Yaskawa INFORM job: R1_W17,20,22(0,0)OK-KMNEW.JBI

/JOB
//NAME R1_W17,20,22(0,0)OK-KMNEW
///FOLDERNAME KRIS-SCIANA
//POS
///NPOS 166,166,0,10,0,0
///TOOL 0
///POSTYPE PULSE
///PULSE
C00000=-143433,-90175,-75020,-14586,83972,33032
C00001=-153732,-78635,-58192,-14050,77869,30109
C00002=-157098,-74863,-52692,-13875,75874,29154
C00003=-157098,-74243,-51213,-13910,75301,29220
C00004=-157098,-74333,-51423,-13906,75382,29211
C00005=-158949,-72964,-50795,-13730,75376,28555
C00006=-157200,-74632,-52271,-13875,75723,29138
C00007=-211231,-129831,-71825,-7304,52478,11413
C00008=-211231,-128371,-70027,-7339,52125,11439
C00009=-211231,-126878,-68176,-7377,51757,11467
C00010=-211231,-127047,-68387,-7373,51799,11463
C00011=-212771,-124423,-67855,-6939,52685,10797
C00012=-211231,-128089,-69679,-7347,52057,11444
C00013=-232444,-132787,-72439,-2403,50152,3160
C00014=-232444,-131349,-70721,-2414,49837,3167
C00015=-232444,-129731,-68771,-2422,49470,3172
C00016=-232444,-129852,-68917,-2422,49498,3172
C00017=-232842,-127642,-68505,-2293,50368,2994
C00018=-232444,-131710,-71149,-2407,49917,3162
C00019=-145968,-32886,-32033,-14386,86409,31863
C00020=-145968,-32298,-29296,-14401,85068,32019
C00021=-145968,-31942,-27784,-14425,84347,32104
C00022=-145968,-31980,-27951,-14410,84425,32095
C00023=-147178,-31176,-27384,-14348,84275,31690
C00024=-145968,-32285,-29241,-14400,85043,32023
C00025=-139425,14039,5691,-14754,88455,33906
C00026=-139519,13379,6497,-14751,87629,33972
C00027=-139519,13616,7680,-14752,87041,34041
C00028=-139519,13563,7430,-14752,87165,34026
C00029=-140335,14099,7919,-14713,86994,33760
C00030=-140218,14798,7500,-14716,87614,33729
C00031=-139869,18363,10790,-14729,87489,33867
C00032=-140218,14798,7500,-14716,87614,33729
C00033=-140402,1849,-19527,-14902,97240,32509
C00034=-140435,1808,-19560,-14885,97235,32499
C00035=-142735,10961,1802,-14568,88645,32727
C00036=-142735,11930,7018,-14580,86016,33037
C00037=-142735,12205,8255,-14585,85414,33107
C00038=-142735,12159,8055,-14585,85510,33096
C00039=-143548,12776,8612,-14541,85338,32830
C00040=-143548,12478,7250,-14533,86001,32752
C00041=-142989,17280,11639,-14579,85875,32965
C00042=-143548,12478,7250,-14533,86001,32752
C00043=-153871,-49826,-39465,-13916,81020,29711
C00044=-153871,-49427,-38150,-13936,80432,29777
C00045=-153871,-48844,-36293,-13969,79619,29871
C00046=-153871,-48918,-36516,-13965,79718,29861
C00047=-155772,-47404,-35637,-13806,79621,29203
C00048=-153871,-49375,-37964,-13941,80356,29788
C00049=-176442,-83720,-50224,-26100,86167,24219
C00050=-176268,-83127,-48832,-26086,85723,24382
C00051=-176268,-82702,-48032,-26088,85476,24434
C00052=-176268,-82805,-48225,-26088,85536,24421
C00053=-177470,-81547,-47714,-26247,85464,23996
C00054=-176268,-83563,-49657,-26078,85980,24323
C00055=-152058,-57095,-47355,-15849,91689,31553
C00056=-147010,-10638,-8183,-21391,105329,31267
C00057=-140743,-13850,-3598,-31425,97214,46819
C00058=-163982,-90504,-45918,-34963,77070,43608
C00059=-165644,-92905,-46739,-35256,75820,43353
C00060=-158551,-98871,-68851,-16167,82483,30472
C00061=-139863,-9121,-22514,-12675,86754,36604
C00062=-142907,-1645,-8358,-12312,81526,36078
C00063=-137448,8074,8661,-24597,77704,52502
C00064=-134515,54764,60771,-29890,95701,49675
C00065=-140743,-13850,-3598,-31425,97214,46819
C00066=-146433,-61661,-62839,-14679,91621,33634
C00067=-152691,-57358,-64796,-14380,93822,31204
C00068=-159687,-62193,-51187,-13527,81199,28324
C00069=-149187,-17486,-8424,-28072,102983,37207
C00070=-171257,-77817,-43106,-31829,86773,32910
C00071=-172558,-79550,-43833,-32051,85919,32654
C00072=-179422,-87952,-47149,-33191,81425,31301
C00073=-188034,-95777,-49870,-34529,76186,29541
C00074=-201576,-85135,-50180,-27119,84644,21010
C00075=-189185,-159173,-100064,-12251,58132,22119
C00076=-139628,-22178,-29745,-13339,88451,36438
C00077=-142464,16713,5801,-14603,90978,35100
C00078=-140096,48315,46031,-21206,94479,42259
C00079=-138998,70596,76957,-24600,99628,41883
C00080=-149221,-17459,-8404,-28081,102973,37195
C00081=-142912,-78923,-74681,-14594,91271,34909
C00082=96,-41537,-55485,-8102,54341,61135
C00083=96,-41537,-55485,-8102,54341,61135
C00084=-47991,-26757,-28892,6367,80786,-11975
C00085=-57126,-9114,2182,8032,71615,-15703
C00086=-56289,-5858,6360,8073,70774,-15813
C00087=-54160,-1963,12621,8049,68923,-15724
C00088=-54160,-1355,14168,8081,68290,-15768
C00089=-54160,-1431,13975,8077,68369,-15762
C00090=-53417,516,15594,7965,68299,-15502
C00091=-53699,-1671,12330,7961,69203,-15542
C00092=-56482,3777,16911,8368,69462,-16522
C00093=-53699,-1671,12330,7961,69203,-15542
C00094=-16096,-40309,-15630,1558,64307,-2146
C00095=-15667,-39835,-14323,1484,63739,-1996
C00096=-15667,-38980,-12408,1491,63001,-2002
C00097=-15667,-39089,-12651,1491,63095,-2002
C00098=-15228,-35710,-10538,1402,63524,-1836
C00099=-15475,-38012,-12587,1447,63607,-1924
C00100=26525,-36306,-13799,-6251,66511,13302
C00101=27157,-34792,-10896,-6403,65558,13584
C00102=27157,-34039,-9183,-6437,64895,13622
C00103=27157,-34142,-9408,-6432,64981,13617
C00104=26710,-32142,-8110,-6346,65173,13444
C00105=27121,-34968,-11568,-6383,65877,13555
C00106=38673,-31750,-14829,-8018,70533,17427
C00107=38106,-27047,-6323,-8075,67686,17416
C00108=38106,-26024,-3889,-8132,66720,17484
C00109=38106,-26093,-4052,-8129,66783,17480
C00110=37587,-24395,-2874,-8044,66879,17284
C00111=38095,-27443,-7349,-8055,68105,17383
C00112=33691,-40237,-37529,-4343,78333,9389
C00113=4088,-38479,-36421,-4266,78531,9229
C00114=6240,-59965,-30493,-1746,62990,4256
C00115=6240,-59198,-28889,-1752,62394,4263
C00116=6240,-59277,-29056,-1752,62455,4263
C00117=6137,-57545,-28162,-1726,62793,4220
C00118=6137,-58794,-30830,-1711,63793,4205
C00119=1139,-59118,-30998,-730,63654,2372
C00120=6137,-58794,-30830,-1711,63793,4205
C00121=47807,-38519,-19261,-8869,69876,19011
C00122=47539,-37304,-17377,-8859,69317,18957
C00123=47539,-36567,-15561,-8901,68588,19011
C00124=47539,-36658,-15781,-8894,68676,19004
C00125=47029,-35461,-15018,-8811,68766,18813
C00126=47893,-38902,-19858,-8871,70056,19027
C00127=73069,7126,14309,-11765,75874,27473
C00128=72335,9424,18352,-11759,74488,27349
C00129=72335,9956,19820,-11792,73873,27410
C00130=72335,9884,19621,-11787,73955,27403
C00131=71491,11415,20993,-11706,73779,27121
C00132=71657,3792,9684,-11575,76785,26891
C00133=61085,-36100,-21666,6391,58079,18912
C00134=49069,-45805,-25229,-7304,68786,15386
C00135=19871,-63611,-22023,35378,44606,-3365
C00136=17766,-52406,-14755,34280,50845,-2144
C00137=56335,-20769,8067,22753,38631,7110
C00138=59032,-16534,11142,20917,38204,8486
C00139=60031,-14754,12465,20223,38057,9000
C00140=61085,-36100,-21666,6391,58079,18912
C00141=29040,-81101,-50034,-3867,64562,8354
C00142=7217,-74366,-42042,361,62632,377
C00143=-16654,-66617,-25209,25593,50854,-13543
C00144=-27368,-47601,-12216,38001,70169,-15327
C00145=17766,-52406,-14755,34280,50845,-2144
C00146=46390,-61269,-41061,-6756,70352,14356
C00147=42236,-65961,-43421,-6101,69070,12939
C00148=21298,-49858,-1802,32067,40583,-8230
C00149=20826,-44930,4480,33075,39613,-8917
C00150=60671,-13467,25003,8839,33164,11366
C00151=62121,-10887,26961,7730,33147,12189
C00152=66302,-2318,33759,4536,33070,14551
C00153=69057,3829,38920,2429,32943,16104
C00154=60086,17396,47844,26002,45227,9224
C00155=60912,19537,49876,25778,44850,9513
C00156=60912,14444,39766,24345,48130,10454
C00157=78652,23072,35845,-11228,70256,25748
C00158=41637,-60211,-42225,-5828,71489,12454
C00159=-9438,-58348,-23745,3601,60262,-5968
C00160=-15357,-59811,-7616,12634,36711,-18275
C00161=-36406,-36757,8811,38530,63422,-26409
C00162=20826,-44930,4480,33075,39613,-8917
C00163=27379,-50240,-5351,20739,41756,-1745
C00164=50643,-51074,-27069,-7729,67873,16514
C00165=-88506,-94181,-91931,-709,81235,59832
BC00000=335653,8129,711615
BC00001=335653,8129,711615
BC00002=335653,8129,711615
BC00003=335653,8129,711615
BC00004=335653,8129,711615
BC00005=335653,8129,711615
BC00006=335653,8129,711615
BC00007=335653,8130,711613
BC00008=335653,8130,711613
BC00009=335653,8130,711613
BC00010=335653,8130,711613
BC00011=335653,8130,711613
BC00012=335653,8130,711613
BC00013=335653,1154,711613
BC00014=335653,1155,711613
BC00015=335653,1155,711613
BC00016=335653,1155,711613
BC00017=335653,1155,711613
BC00018=335653,1155,711613
BC00019=335653,1154,711612
BC00020=335653,1154,711612
BC00021=335653,1154,711612
BC00022=335653,1154,711612
BC00023=335653,1154,711612
BC00024=335653,1154,711612
BC00025=335653,1152,711610
BC00026=335653,1152,711610
BC00027=335653,1152,711610
BC00028=335653,1152,711610
BC00029=335653,1152,711610
BC00030=335653,1152,711610
BC00031=335653,1152,711610
BC00032=335653,1152,711610
BC00033=335653,1152,711610
BC00034=160380,1151,711608
BC00035=160380,1151,715049
BC00036=160380,1151,715049
BC00037=160380,1151,715049
BC00038=160380,1151,715049
BC00039=160380,1151,715049
BC00040=160380,1151,715049
BC00041=160380,1152,715048
BC00042=160380,1151,715049
BC00043=160380,1151,715049
BC00044=160380,1151,715049
BC00045=160380,1151,715049
BC00046=160380,1151,715049
BC00047=160380,1151,715049
BC00048=160380,1151,715049
BC00049=160380,1151,715049
BC00050=160380,1151,715049
BC00051=160380,1151,715049
BC00052=160380,1151,715049
BC00053=160380,1151,715049
BC00054=160380,1151,715049
BC00055=160380,1151,715049
BC00056=160380,1151,715049
BC00057=160380,1151,715049
BC00058=160380,1151,715049
BC00059=160380,1151,715049
BC00060=160381,1151,715048
BC00061=160381,1151,715048
BC00062=160381,1151,715048
BC00063=160382,1151,715048
BC00064=160382,1151,715048
BC00065=160380,1151,715049
BC00066=160381,1151,715048
BC00067=347379,1151,715048
BC00068=347379,1151,715048
BC00069=347378,1151,715047
BC00070=347378,1151,715047
BC00071=347378,1151,715047
BC00072=347378,1151,715046
BC00073=347378,1151,715046
BC00074=347378,1151,715046
BC00075=347379,1151,715048
BC00076=347379,1151,715048
BC00077=347379,1151,715048
BC00078=347378,1151,715047
BC00079=347378,1151,715047
BC00080=347378,1151,715047
BC00081=347379,1151,715048
BC00082=71294,1151,1035267
BC00083=71294,1151,1035267
BC00084=14908,77377,861464
BC00085=14908,77377,833834
BC00086=14908,77377,833863
BC00087=14909,77377,833909
BC00088=14909,77377,833909
BC00089=14909,77377,833909
BC00090=14909,77377,833909
BC00091=14909,77377,833909
BC00092=14909,77377,833909
BC00093=14909,77377,833909
BC00094=14909,77377,833909
BC00095=14909,77377,833909
BC00096=14909,77376,833908
BC00097=14909,77376,833908
BC00098=14909,77376,833908
BC00099=14909,77376,833908
BC00100=14909,77376,833908
BC00101=14909,77376,833908
BC00102=14909,77376,833908
BC00103=14909,77376,833908
BC00104=14909,77376,833908
BC00105=14909,77376,833908
BC00106=14909,77376,833908
BC00107=14909,77376,833908
BC00108=14909,77376,833907
BC00109=14909,77376,833907
BC00110=14909,77376,833907
BC00111=14909,77376,833907
BC00112=14908,77377,833834
BC00113=166638,196652,833834
BC00114=218128,196652,810863
BC00115=218128,196652,810863
BC00116=218128,196652,810863
BC00117=218128,196652,810863
BC00118=218128,196652,810863
BC00119=218128,196652,810863
BC00120=218128,196652,810863
BC00121=218128,196652,810863
BC00122=218128,196652,810863
BC00123=218128,196652,810863
BC00124=218128,196652,810863
BC00125=218128,196652,810863
BC00126=218128,196652,810863
BC00127=218127,196651,810862
BC00128=218127,196651,810862
BC00129=218127,196651,810862
BC00130=218127,196651,810862
BC00131=218127,196651,810862
BC00132=218127,196651,810862
BC00133=218128,196652,810863
BC00134=218128,196652,810863
BC00135=218128,196652,810863
BC00136=218128,196652,810863
BC00137=218128,196652,810863
BC00138=218128,196652,810863
BC00139=218128,196652,810863
BC00140=218128,196652,810863
BC00141=218128,196652,810863
BC00142=218128,196652,810863
BC00143=218128,196652,810863
BC00144=218128,196652,810863
BC00145=218128,196652,810863
BC00146=218128,196652,810863
BC00147=35771,188457,887876
BC00148=35771,188457,887876
BC00149=35771,188457,887876
BC00150=35771,188457,887876
BC00151=35771,188457,887876
BC00152=35771,188457,887876
BC00153=35771,188457,887876
BC00154=35771,188457,887876
BC00155=35771,188457,887876
BC00156=35771,188457,887876
BC00157=35772,185483,887872
BC00158=35772,185483,887872
BC00159=35772,185483,887872
BC00160=35771,188457,887876
BC00161=35771,188457,887876
BC00162=35771,188457,887876
BC00163=36231,187575,887592
BC00164=38104,183984,886436
BC00165=294911,15771,909309
///POSTYPE BASE
///RECTAN
///RCONF 0,0,0,0,1,0,0,0,0,0,0,0,0,0,0,0,0,0,0,0,0,0,0,0
P00006=2.006,1.622,-0.565,0.0000,0.0000,0.0000
P00021=0.073,2.058,-0.109,0.0000,0.0000,0.0000
P00022=2.006,1.622,-0.565,0.0000,0.0000,0.0000
///RCONF 0,0,0,0,0,0,0,0,0,0,0,0,0,0,0,0,0,0,0,0,0,0,0,0
P00023=-2.957,-4.083,2.762,0.0000,0.0000,0.0000
P00024=-1.466,-0.226,-0.419,0.0000,0.0000,0.0000
P00025=3.643,0.007,-2.585,0.0000,0.0000,0.0000
P00026=2.644,0.055,-2.583,0.0000,0.0000,0.0000
P00027=2.278,0.099,-4.210,0.0000,0.0000,0.0000
P00028=-1.778,-0.182,-2.050,0.0000,0.0000,0.0000
P00029=1.749,4.006,-0.261,0.0000,0.0000,0.0000
//INST
///DATE 2025/04/16 06:31
///ATTR SC,RW
///GROUP1 RB1,BS1
///LVARS 0,1,0,0,0,2,2,0
NOP
MOVJ C00000 BC00000 VJ=50.00
SFTOF
MOVL C00001 BC00001 V=333.3
MOVL C00002 BC00002 V=166.7
REFP 3 C00003 BC00003
CALL JOB:SEARCH-R1
SET P021 P006
SFTON P021
MOVL C00004 BC00004 V=60.0
REFP 3 C00005 BC00005
CALL JOB:SEARCH-R1
SET P021 P006
SFTON P021
MOVL C00006 BC00006 V=166.7
MOVL C00007 BC00007 V=500.0
MOVL C00008 BC00008 V=166.7
REFP 3 C00009 BC00009
CALL JOB:SEARCH-R1
SET P022 P006
SFTON P022
MOVL C00010 BC00010 V=60.0
REFP 3 C00011 BC00011
CALL JOB:SEARCH-R1
SET P022 P006
SFTON P022
MOVL C00012 BC00012 V=166.7
MOVL C00013 BC00013 V=500.0
MOVL C00014 BC00014 V=166.7
REFP 3 C00015 BC00015
CALL JOB:SEARCH-R1
SET P023 P006
SFTON P023
MOVL C00016 BC00016 V=60.0
REFP 3 C00017 BC00017
CALL JOB:SEARCH-R1
SET P023 P006
SFTON P023
MOVL C00018 BC00018 V=166.7
MOVL C00019 BC00019 V=500.0
MOVL C00020 BC00020 V=166.7
REFP 3 C00021 BC00021
CALL JOB:SEARCH-R1
SET P024 P006
SFTON P024
MOVL C00022 BC00022 V=60.0
REFP 3 C00023 BC00023
CALL JOB:SEARCH-R1
SET P024 P006
SFTON P024
MOVL C00024 BC00024 V=166.7
MOVL C00025 BC00025 V=500.0
MOVL C00026 BC00026 V=166.7
REFP 3 C00027 BC00027
CALL JOB:SEARCH-R1
SET P025 P006
SFTON P025
MOVL C00028 BC00028 V=60.0
REFP 3 C00029 BC00029
CALL JOB:SEARCH-R1
SET P025 P006
SFTON P025
MOVL C00030 BC00030 V=166.7
REFP 3 C00031 BC00031
CALL JOB:SEARCH-R1
SET P025 P006
SFTON P025
MOVL C00032 BC00032 V=166.7
SFTOF
MOVL C00033 BC00033 V=500.0
MOVL C00034 BC00034 V=500.0
MOVL C00035 BC00035 V=500.0
MOVL C00036 BC00036 V=166.7
REFP 3 C00037 BC00037
CALL JOB:SEARCH-R1
SET P026 P006
SFTON P026
MOVL C00038 BC00038 V=60.0
REFP 3 C00039 BC00039
CALL JOB:SEARCH-R1
SET P026 P006
SFTON P026
MOVL C00040 BC00040 V=166.7
REFP 3 C00041 BC00041
CALL JOB:SEARCH-R1
SET P026 P006
SFTON P026
MOVL C00042 BC00042 V=166.7
MOVL C00043 BC00043 V=500.0
MOVL C00044 BC00044 V=166.7
REFP 3 C00045 BC00045
CALL JOB:SEARCH-R1
SET P027 P006
SFTON P027
MOVL C00046 BC00046 V=60.0
REFP 3 C00047 BC00047
CALL JOB:SEARCH-R1
SET P027 P006
SFTON P027
MOVL C00048 BC00048 V=166.7
MOVL C00049 BC00049 V=500.0
MOVL C00050 BC00050 V=166.7
REFP 3 C00051 BC00051
CALL JOB:SEARCH-R1
SET P028 P006
SFTON P028
MOVL C00052 BC00052 V=60.0
REFP 3 C00053 BC00053
CALL JOB:SEARCH-R1
SET P028 P006
SFTON P028
MOVL C00054 BC00054 V=166.7
SFTOF
MOVL C00055 BC00055 V=166.7
CALL JOB:COFNIJ_DRUT
MACRO1 MJ#(0) ARGF9
MOVL C00056 BC00056 V=500.0
SFTON P027
MOVL C00057 BC00057 V=166.7 PL=0
ARCON
SFTON P028
MOVL C00058 BC00058 V=12.5
MOVL C00059 BC00059 V=12.5
ARCOF
SFTOF
MOVJ C00060 BC00060 VJ=25.00
MOVJ C00061 BC00061 VJ=25.00
MOVJ C00062 BC00062 VJ=25.00
SFTON P026
MOVL C00063 BC00063 V=166.7 PL=0
ARCON
MOVL C00064 BC00064 V=12.5
SFTON P027
MOVL C00065 BC00065 V=12.5
ARCOF
SFTOF
MOVJ C00066 BC00066 VJ=25.00
MOVJ C00067 BC00067 VJ=25.00
MOVJ C00068 BC00068 VJ=25.00
SFTON P021
MOVL C00069 BC00069 V=166.7 PL=0
ARCON
SFTON P022
MOVL C00070 BC00070 V=12.5
MOVL C00071 BC00071 V=12.5
ARCOF
SFTON P023
MOVL C00072 BC00072 V=41.7 PL=0
ARCON
MOVL C00073 BC00073 V=12.5
MOVL C00074 BC00074 V=12.5
ARCOF
SFTOF
MOVJ C00075 BC00075 VJ=25.00
MOVJ C00076 BC00076 VJ=25.00
MOVJ C00077 BC00077 VJ=25.00
SFTON P024
MOVL C00078 BC00078 V=166.7 PL=0
ARCON
MOVL C00079 BC00079 V=12.5
SFTON P021
MOVL C00080 BC00080 V=12.5
ARCOF
SFTOF
MOVJ C00081 BC00081 VJ=25.00
MOVJ C00082 BC00082 VJ=25.00
CALL JOB:CLEAN-R1_LONG
MOVJ C00083 BC00083 VJ=25.00
MOVJ C00084 BC00084 VJ=25.00
MOVJ C00085 BC00085 VJ=25.00
MOVL C00086 BC00086 V=500.0
MOVL C00087 BC00087 V=166.7
REFP 3 C00088 BC00088
CALL JOB:SEARCH-R1
SET P021 P006
SFTON P021
MOVL C00089 BC00089 V=60.0
REFP 3 C00090 BC00090
CALL JOB:SEARCH-R1
SET P021 P006
SFTON P021
MOVL C00091 BC00091 V=166.7
REFP 3 C00092 BC00092
CALL JOB:SEARCH-R1
SET P025 P006
SFTON P025
MOVL C00093 BC00093 V=166.7
SFTON P021
MOVL C00094 BC00094 V=500.0
MOVL C00095 BC00095 V=166.7
REFP 3 C00096 BC00096
CALL JOB:SEARCH-R1
SET P022 P006
SFTON P022
MOVL C00097 BC00097 V=60.0
REFP 3 C00098 BC00098
CALL JOB:SEARCH-R1
SET P022 P006
SFTON P022
MOVL C00099 BC00099 V=166.7
MOVL C00100 BC00100 V=500.0
MOVL C00101 BC00101 V=166.7
REFP 3 C00102 BC00102
CALL JOB:SEARCH-R1
SET P023 P006
SFTON P023
MOVL C00103 BC00103 V=60.0
REFP 3 C00104 BC00104
CALL JOB:SEARCH-R1
SET P023 P006
SFTON P023
MOVL C00105 BC00105 V=166.7
MOVL C00106 BC00106 V=500.0
MOVL C00107 BC00107 V=166.7
REFP 3 C00108 BC00108
CALL JOB:SEARCH-R1
SET P024 P006
SFTON P024
MOVL C00109 BC00109 V=60.0
REFP 3 C00110 BC00110
CALL JOB:SEARCH-R1
SET P024 P006
SFTON P024
MOVL C00111 BC00111 V=166.7
SFTOF
MOVL C00112 BC00112 V=500.0
MOVL C00113 BC00113 V=500.0
MOVL C00114 BC00114 V=166.7
REFP 3 C00115 BC00115
CALL JOB:SEARCH-R1
SET P026 P006
SFTON P026
MOVL C00116 BC00116 V=60.0
REFP 3 C00117 BC00117
CALL JOB:SEARCH-R1
SET P026 P006
SFTON P026
MOVL C00118 BC00118 V=166.7
REFP 3 C00119 BC00119
CALL JOB:SEARCH-R1
SET P027 P006
SFTON P027
MOVL C00120 BC00120 V=166.7
SFTON P026
MOVL C00121 BC00121 V=500.0
MOVL C00122 BC00122 V=166.7
REFP 3 C00123 BC00123
CALL JOB:SEARCH-R1
SET P028 P006
SFTON P028
MOVL C00124 BC00124 V=60.0
REFP 3 C00125 BC00125
CALL JOB:SEARCH-R1
SET P028 P006
SFTON P028
MOVL C00126 BC00126 V=166.7
MOVL C00127 BC00127 V=500.0
MOVL C00128 BC00128 V=166.7
REFP 3 C00129 BC00129
CALL JOB:SEARCH-R1
SET P029 P006
SFTON P029
MOVL C00130 BC00130 V=60.0
REFP 3 C00131 BC00131
CALL JOB:SEARCH-R1
SET P029 P006
SFTON P029
MOVL C00132 BC00132 V=166.7
SFTOF
MOVL C00133 BC00133 V=166.7
CALL JOB:COFNIJ_DRUT
MACRO1 MJ#(0) ARGF9
SFTON P028
MOVL C00134 BC00134 V=500.0
MOVL C00135 BC00135 V=500.0
MOVL C00136 BC00136 V=166.7 PL=0
ARCON
SFTON P029
MOVL C00137 BC00137 V=12.5
MOVL C00138 BC00138 V=12.5
MOVL C00139 BC00139 V=12.5
ARCOF
SFTOF
MOVJ C00140 BC00140 VJ=25.00
MOVJ C00141 BC00141 VJ=25.00
MOVJ C00142 BC00142 VJ=25.00
SFTON P027
MOVL C00143 BC00143 V=166.7 PL=0
ARCON
SFTON P026
MOVL C00144 BC00144 V=12.5
SFTON P028
MOVL C00145 BC00145 V=12.5
ARCOF
SFTOF
MOVJ C00146 BC00146 VJ=25.00
MOVJ C00147 BC00147 VJ=25.00
MOVJ C00148 BC00148 VJ=25.00
SFTON P022
MOVL C00149 BC00149 V=166.7 PL=0
ARCON
SFTON P023
MOVL C00150 BC00150 V=12.5
MOVL C00151 BC00151 V=12.5
ARCOF
SFTON P024
MOVL C00152 BC00152 V=41.7 PL=0
ARCON
MOVL C00153 BC00153 V=12.5
MOVL C00154 BC00154 V=12.5
MOVL C00155 BC00155 V=12.5
ARCOF
MOVL C00156 BC00156 V=166.7
SFTOF
MOVJ C00157 BC00157 VJ=25.00
MOVJ C00158 BC00158 VJ=25.00
MOVJ C00159 BC00159 VJ=25.00
SFTON P025
MOVL C00160 BC00160 V=166.7 PL=0
ARCON
SFTON P021
MOVL C00161 BC00161 V=12.5
SFTON P022
MOVL C00162 BC00162 V=12.5
ARCOF
MOVL C00163 BC00163 V=166.7
SFTOF
MOVJ C00164 BC00164 VJ=40.00
MOVJ C00165 BC00165 VJ=40.00
END
